{attribute 'qualified_only'}
VAR_GLOBAL
  //-----------------------------------------------------------------------------------------------------------
  // MB TriggerBox, set output to activate camera, get input timestamp from flash controller
  //-----------------------------------------------------------------------------------------------------------
  MessageLevelTriggerBox      : ARRAY[1..MAX_TRIGGER_BOX] OF E_MessageType; // individual message level for every box.

{IF defined (XFC)}
  TriggerBoxCtrl              : ARRAY[1..MAX_TRIGGER_BOX] OF Fb_TriggerBox;   // execution of trigger function
{ELSE}
  TriggerBoxCtrl              : ARRAY[1..MAX_TRIGGER_BOX] OF I_TriggerBox;   // execution of trigger function
{END_IF}

  TriggerBox                  : ARRAY[1..MAX_TRIGGER_BOX] OF ST_TriggerBox;   // .ToPlc   --> write your commands in here
                                                                    // .FromPlc --> read your results from here

  DigitalOutPutDCState  AT %I*  : ARRAY[1..MAX_TRIGGER_BOX] OF ST_DC_State;

  DigitalOutputDC   AT %Q*      : ARRAY[1..MAX_TRIGGER_BOX] OF ST_DC_Output;
  DigitalInputDC    AT %I*      : ARRAY[1..MAX_TRIGGER_BOX] OF ST_DC_Input; // distributed clock digital input with timestamps positive & negative


  //-----------------------------------------------------------------------------------------------------------
  // MB Touch Probe, get input timestamp within axis window, get prcise position using the timestamp
  //-----------------------------------------------------------------------------------------------------------
  MessageLevelTouchProbe      : ARRAY[1..MAX_TRIGGER_BOX] OF E_MessageType; // individual message level for every touch probe

{IF defined (XFC)}
  TouchProbeCtrl              : ARRAY[1..MAX_TOUCH_PROBE] OF Fb_TouchProbe;   // execution of Touch probe function
{ELSE}
  TouchProbeCtrl              : ARRAY[1..MAX_TOUCH_PROBE] OF I_TouchProbe;   // execution of Touch probe function
{END_IF}

  TouchProbe                  : ARRAY[1..MAX_TOUCH_PROBE] OF ST_TouchProbe;   // .ToPlc   --> write your commands in here
                                                                    // .FromPlc --> read your results from here

  //DigitalInputDC    AT %I*    : ARRAY[1..MAX_TOUCH_PROBE] OF ST_DC_Input; // distributed clock digital input with timestamps positive & negative
  DigitalInput      AT %I*    : ARRAY[1..MAX_TOUCH_PROBE] OF ST_MTI_INPUT;    // multi time stamp, one channel
  DigitalState      AT %I*    : ARRAY[1..MAX_TOUCH_PROBE] OF ST_MTI_STATUS;   // multi time stamp status from terminal

END_VAR

(* stored: Version 1.1.0.1, ProductVersion 3.1.4024.12
   GVL GVL_FUNCTIONS: Id {c671dfde-44dd-4068-bb14-c2c3ee47ab68} *)
